Staubli VAL3: workTabSpd.pgx

program workTabSpd()
  local point l_pCurrent
begin
  //K：num of worktable speed code
  do
    l_pCurrent=here(tPrdTool,fPrdFrame)
    nCurtRadius=sqrt(l_pCurrent.trsf.x*l_pCurrent.trsf.x+l_pCurrent.trsf.y*l_pCurrent.trsf.y)
    //速度分段
    nTabSpdCode=K-roundDown(K*nCurtRadius/nPrdRadius)
    call io:tableSpeed(nTabSpdCode)
  until dioGet(io:doB_9_tableOn)==0 or bCycle==false or date:bWorTbMoving==false
end
